(* PLC project Unnamed, Unknown Unnamed 1 *)
(* stored: creationDateTime 2023-03-10T10:37:17, modificationDateTime 2023-03-15T15:56:42 *)

(* https://www.gds2.de/fileadmin/umwelttechnik/umwelttechnik/skripte/steuerungstechnik_ut_2017.pdf, 2.15 *)
FUNCTION_BLOCK Wind_Direction_Indicator
  VAR_INPUT
    IN1 : BOOL;
    IN2 : BOOL;
    IN3 : BOOL;
  END_VAR
  VAR_OUTPUT
    OUT1 : BOOL;
    OUT2 : BOOL;
    OUT3 : BOOL;
    OUT4 : BOOL;
  END_VAR
  VAR  (* added by the conversion: wires and edge detectors of the diagram *)
    _AND55_OUT : BOOL;
    _AND7_OUT : BOOL;
    _AND27_OUT : BOOL;
    _AND41_OUT : BOOL;
  END_VAR

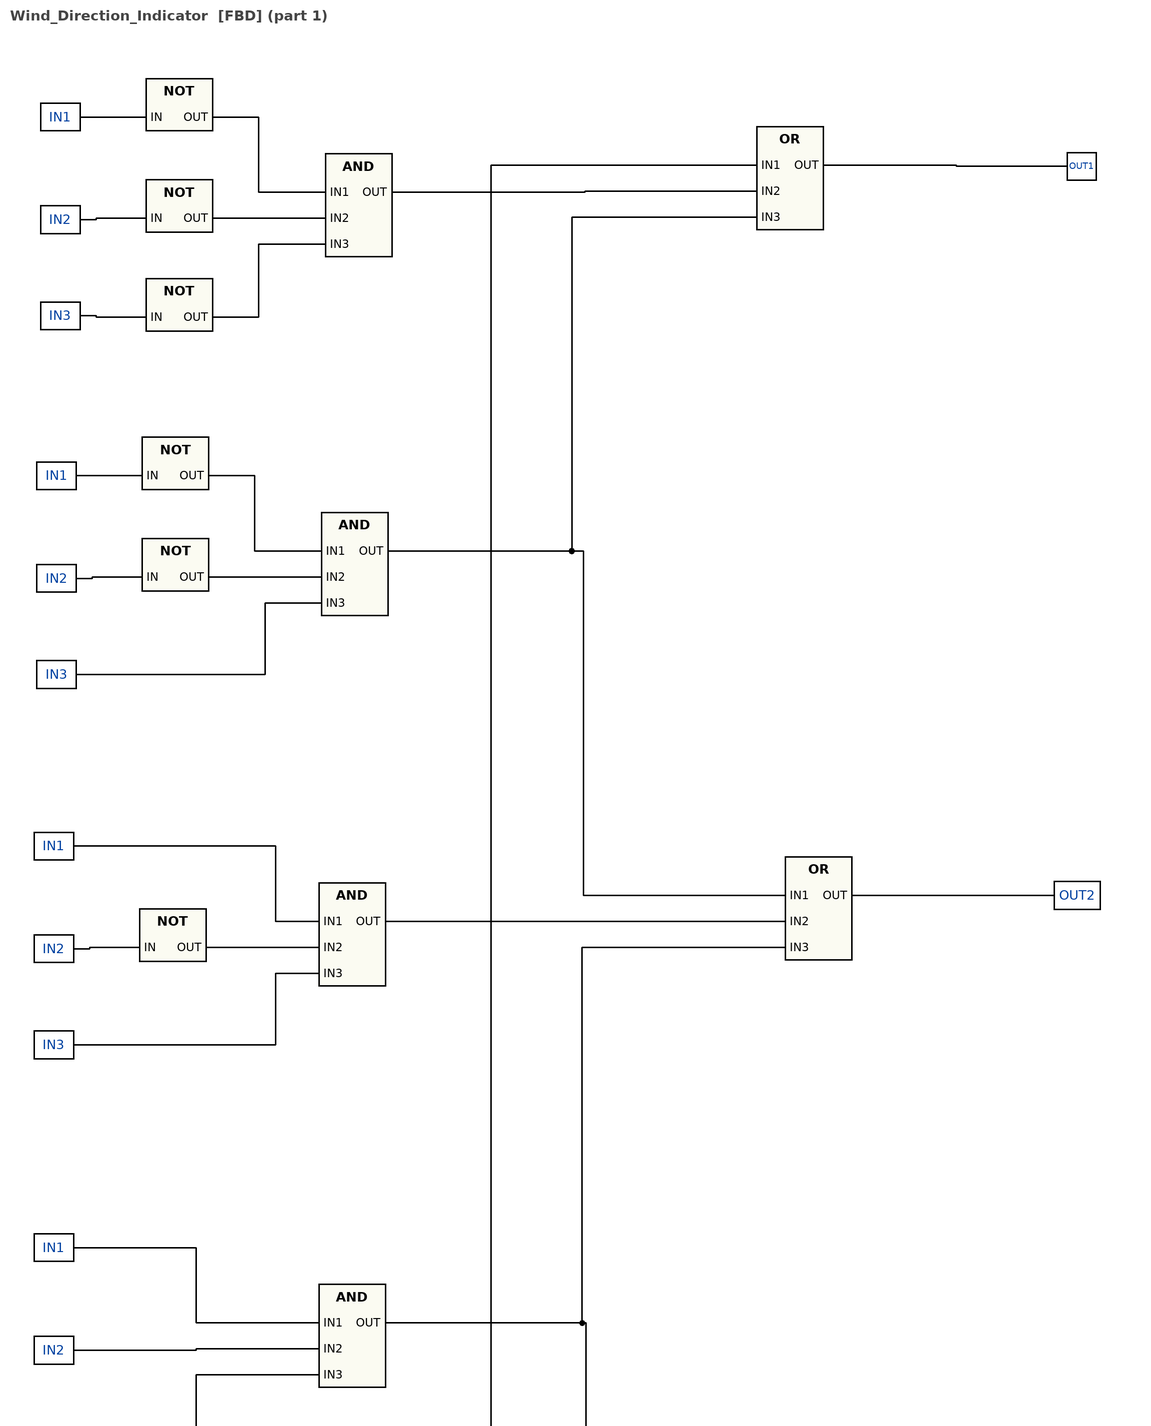
(* FBD diagram, written out as Structured Text *)
_AND55_OUT := IN1 AND NOT IN2 AND NOT IN3;
_AND7_OUT := NOT IN1 AND NOT IN2 AND IN3;
OUT1 := _AND55_OUT OR NOT IN1 AND NOT IN2 AND NOT IN3 OR _AND7_OUT;
_AND27_OUT := IN1 AND IN2 AND IN3;
OUT2 := _AND7_OUT OR IN1 AND NOT IN2 AND IN3 OR _AND27_OUT;
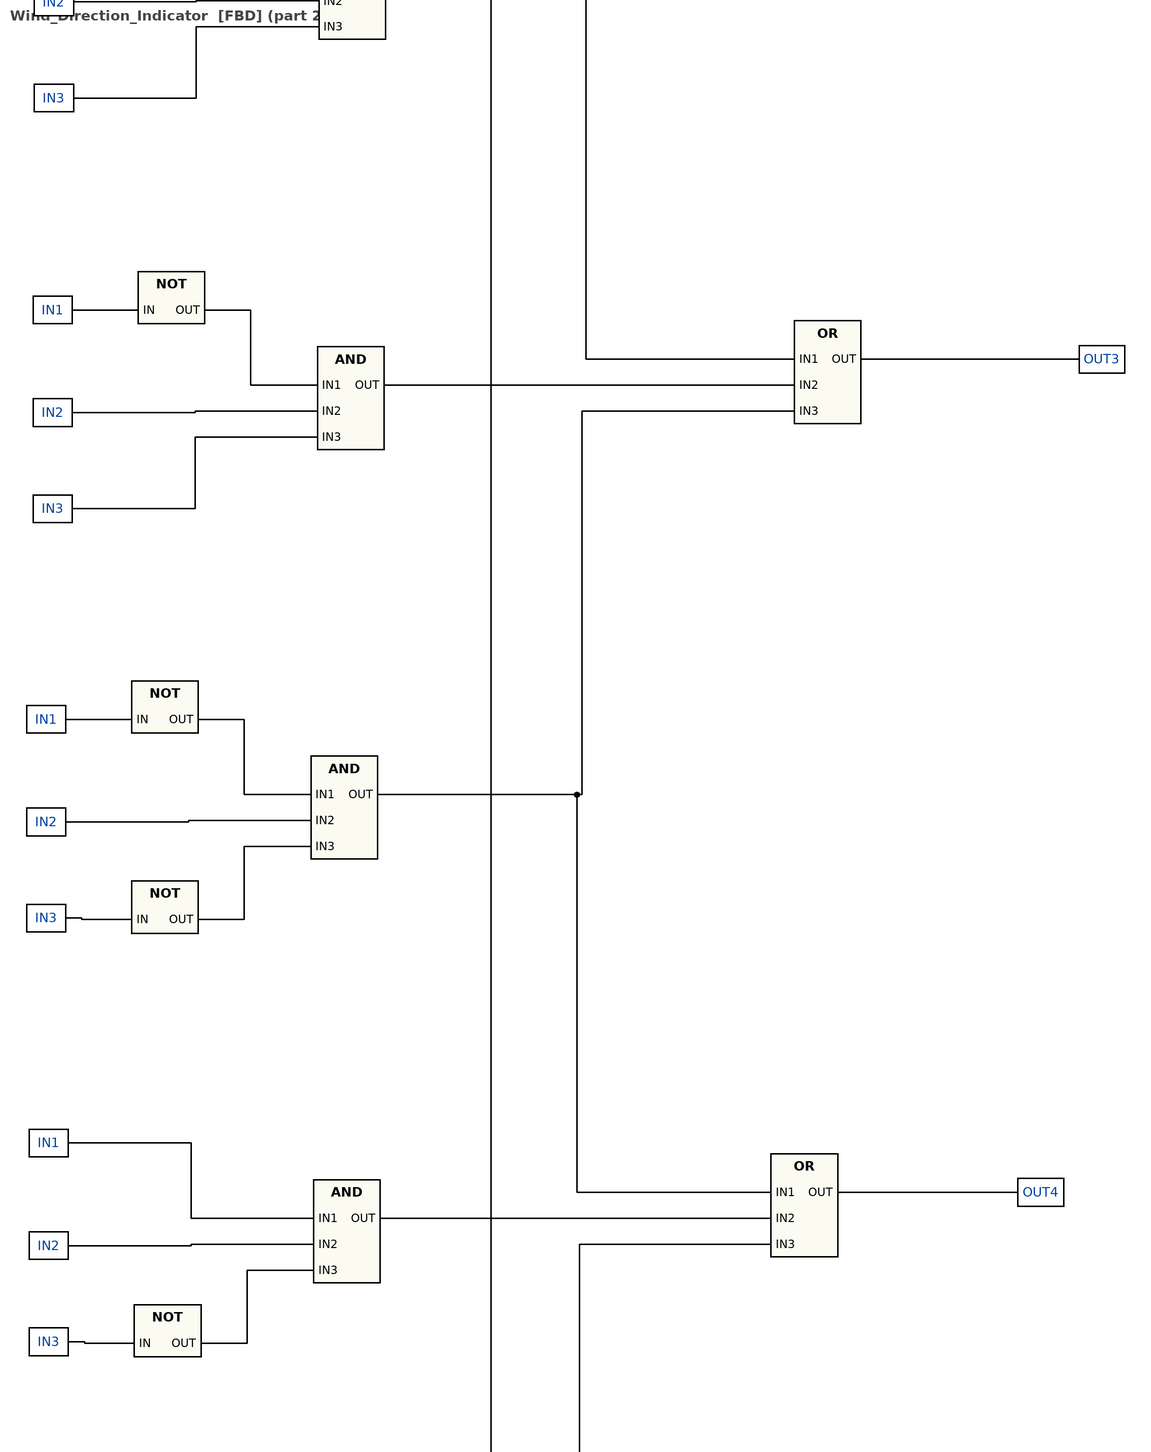
_AND41_OUT := NOT IN1 AND IN2 AND NOT IN3;
OUT3 := _AND27_OUT OR NOT IN1 AND IN2 AND IN3 OR _AND41_OUT;
OUT4 := _AND41_OUT OR IN1 AND IN2 AND NOT IN3 OR _AND55_OUT;
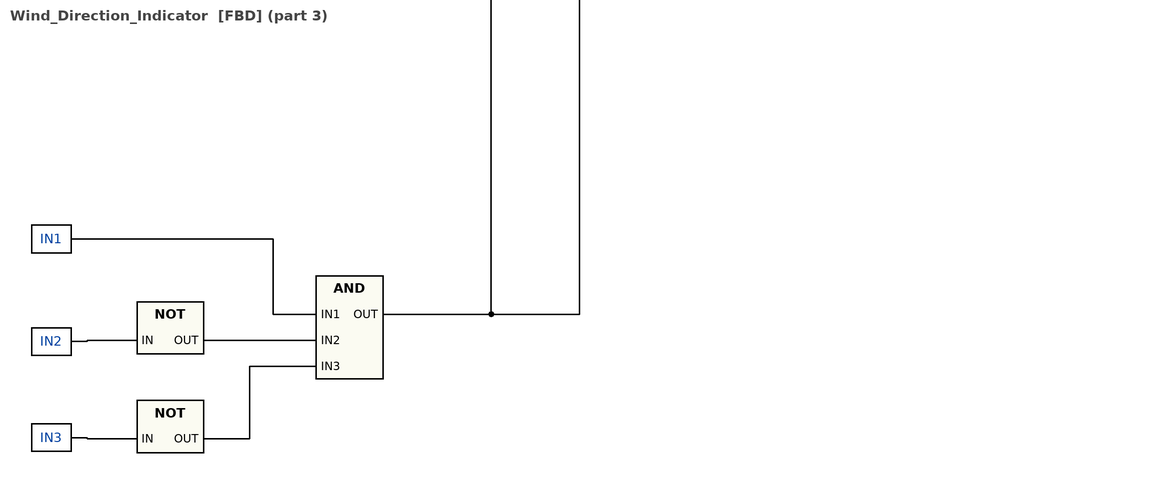
END_FUNCTION_BLOCK

CONFIGURATION config
  RESOURCE resource1 ON PLC
  END_RESOURCE
END_CONFIGURATION
